// TIA Portal project "hognphuongtram3" (V16)

(* hardware
DEVICE "S7-1200 station_1"  S7-1200 Station
   slot 0: "Rack_0"  S7-1200 Rack  Rack  V1.0
   slot 1: "PLC_1"  CPU 1212C DC/DC/DC  6ES7 212-1AE40-0XB0  V4.3
   slot 2: "DI 16/DQ 16x24VDC_1"  6ES7 223-1BL32-0XB0  V2.0
   slot 3: "DQ 16xRelay_1"  SM 1222 DQ16 x relay  6ES7 222-1HH32-0XB0  V2.0
*)

// ===== PLC "PLC_1"  CPU 1212C DC/DC/DC =====

VAR_GLOBAL   // PLC tag table "Default tag table"
   "Tag_1" AT %I0.5 : Bool;
   "KM1" AT %Q0.0 : Bool;
   "Tag_3" AT %I0.0 : Bool;
   "Tag_4" AT %M0.1 : Bool;
   "Tag_5" AT %M0.2 : Bool;
   "Tag_6" AT %M0.3 : Bool;
   "Tag_7" AT %I0.1 : Bool;
   "Tag_8" AT %I0.2 : Bool;
   "Tag_9" AT %M0.4 : Bool;
   "Tag_10" AT %I0.3 : Bool;
   "Tag_11" AT %M0.5 : Bool;
   "Tag_12" AT %I0.4 : Bool;
   "Tag_13" AT %M0.6 : Bool;
   "start" AT %I1.3 : Bool;
   "stop" AT %I1.2 : Bool;
   "Tag_16" AT %I0.6 : Bool;
   "Tag_17" AT %I0.7 : Bool;
   "Tag_18" AT %I1.0 : Bool;
   "Tag_19" AT %I1.1 : Bool;
   "KM2" AT %Q0.1 : Bool;
   "KM3" AT %Q0.2 : Bool;
   "KM4" AT %Q0.3 : Bool;
   "KM5" AT %Q0.4 : Bool;
END_VAR

ORGANIZATION_BLOCK "Main"   // OB1, LAD, ProgramCycle
TITLE = "Main Program Sweep (Cycle)"
{ S7_Optimized_Access := 'TRUE' }
VERSION : 0.1
   VAR_INPUT
      Initial_Call : Bool;   // Initial call of this OB
      Remanence : Bool;   // =True, if remanent data are available
   END_VAR
BEGIN

REGION Network 1
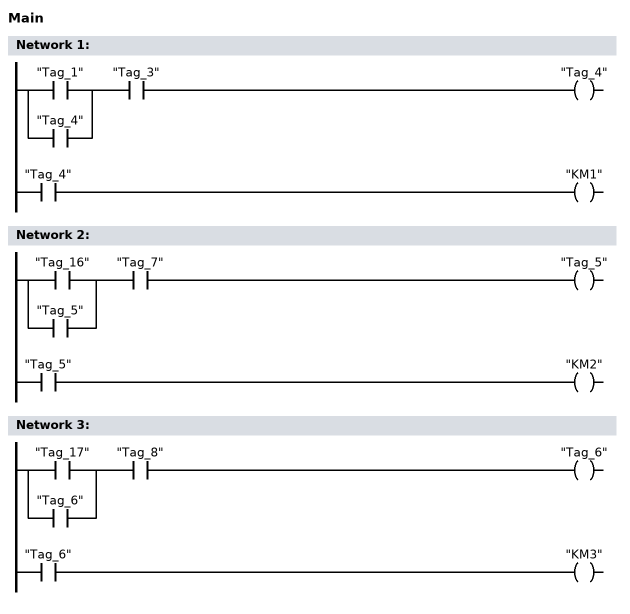
   RUNG wire#powerrail
      Contact( "Tag_1" )
      wire#w1
      Contact( "Tag_3" )
      Coil( "Tag_4" )
   END_RUNG
   RUNG wire#powerrail
      Contact( "Tag_4" )
   END_RUNG wire#w1
   RUNG wire#powerrail
      Contact( "Tag_4" )
      Coil( "KM1" )
   END_RUNG
   // the same network as SCL:
   "Tag_4" := ("Tag_1" OR "Tag_4") AND "Tag_3";
   "KM1" := "Tag_4";
END_REGION

REGION Network 2
   RUNG wire#powerrail
      Contact( "Tag_16" )
      wire#w1
      Contact( "Tag_7" )
      Coil( "Tag_5" )
   END_RUNG
   RUNG wire#powerrail
      Contact( "Tag_5" )
   END_RUNG wire#w1
   RUNG wire#powerrail
      Contact( "Tag_5" )
      Coil( "KM2" )
   END_RUNG
   // the same network as SCL:
   "Tag_5" := ("Tag_16" OR "Tag_5") AND "Tag_7";
   "KM2" := "Tag_5";
END_REGION

REGION Network 3
   RUNG wire#powerrail
      Contact( "Tag_17" )
      wire#w1
      Contact( "Tag_8" )
      Coil( "Tag_6" )
   END_RUNG
   RUNG wire#powerrail
      Contact( "Tag_6" )
   END_RUNG wire#w1
   RUNG wire#powerrail
      Contact( "Tag_6" )
      Coil( "KM3" )
   END_RUNG
   // the same network as SCL:
   "Tag_6" := ("Tag_17" OR "Tag_6") AND "Tag_8";
   "KM3" := "Tag_6";
END_REGION
END_ORGANIZATION_BLOCK